(* Logix 5000 project; controller lab_1 vendor 1 type 14 code 96 rev 28.11; software revision 28.00 *)

TASK MainTask (continuous, watchdog 500 ms) : MainProgram

MODULES
   Local : vendor 1 type 14 code 96 (ICP 1, rev 28.11)
      INPUT : vendor 1 type 7 code 2 (ICP 2, rev 3.1, Input RPI 20 ms)
      RELAY_4 : 1756-OW16I (ICP 4, rev 3.1, Output RPI 20 ms)
      Relay_1 : 1756-OW16I (ICP 0, rev 3.3, Output RPI 20 ms)
      Relay_8 : 1756-IF6I (ICP 6, rev 1.1, Input RPI 100 ms)
      Relay_7 : vendor 1 type 10 code 4 (ICP 5, rev 1.12, Output RPI 25 ms)
END_MODULES

PROGRAM MainProgram   (* main routine MainRoutine *)
VAR
   BAND_01 : FBD_BOOLEAN_AND := (In1 := 1, In2 := 1, In3 := 1, In4 := 1, In5 := 1, In6 := 1, In7 := 1, In8 := 1);
   BOR_01 : FBD_BOOLEAN_OR;
   ESTOP : ALIAS FOR Local:2:I.Data.8;
   RED_LIGHT : ALIAS FOR Local:4:O.Data.2;
   run : BOOL;
   RUN_CMD : BOOL;
   START : ALIAS FOR Local:2:I.Data.0;
   STOP : ALIAS FOR Local:2:I.Data.9;
END_VAR

ROUTINE FBD_Motor_Control   (* function block diagram *)
   SHEET 1
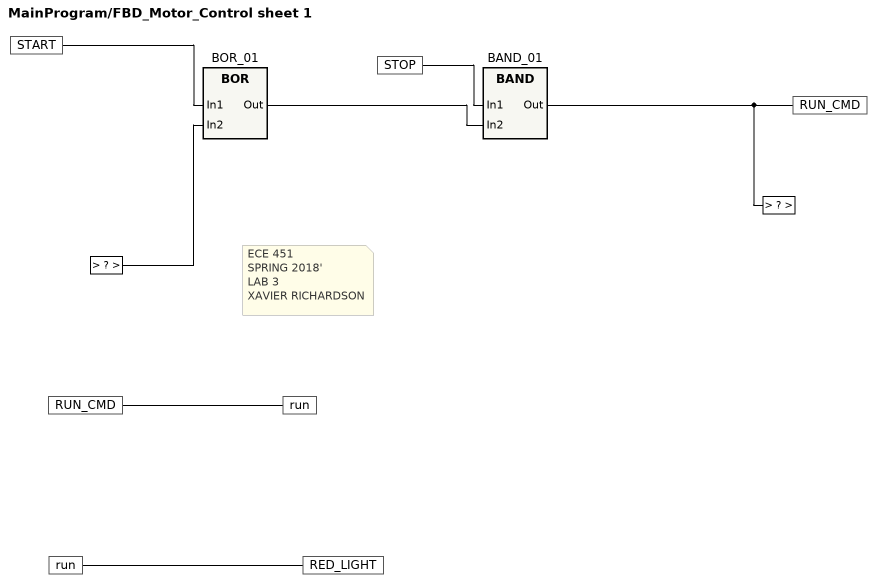
   // ECE 451
   // SPRING 2018'
   // LAB 3
   // XAVIER RICHARDSON
   BOR_01 : BOR(In1 := START, In2 := WIRE(?) {feedback});
   run := RUN_CMD;
   RED_LIGHT := run;
   BAND_01 : BAND(In1 := STOP, In2 := BOR_01.Out);
   WIRE(?) := BAND_01.Out;
   RUN_CMD := BAND_01.Out;
END_ROUTINE

ROUTINE MainRoutine   (* ladder *)
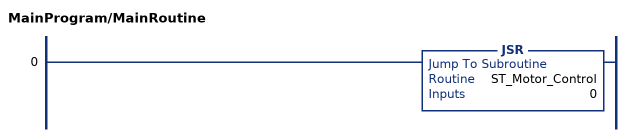
   0: JSR(ST_Motor_Control,0);
END_ROUTINE

ROUTINE Motor_Control   (* ladder *)
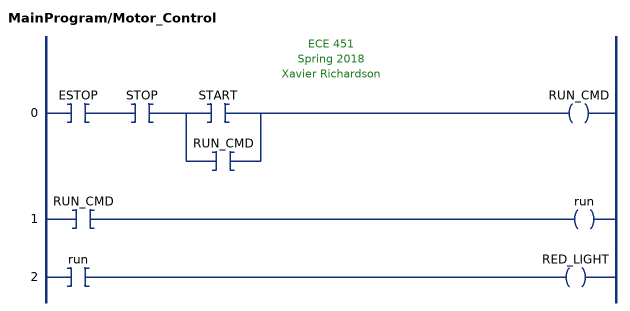
   // ECE 451
   // Spring 2018
   // Xavier Richardson
   0: XIC(ESTOP)XIC(STOP)[XIC(START) ,XIC(RUN_CMD) ]OTE(RUN_CMD);
   1: XIC(RUN_CMD)OTE(run);
   2: XIC(run)OTE(RED_LIGHT);
END_ROUTINE

ROUTINE ST_Motor_Control   (* structured text *)
   (*
   ECE 451 SPRING 2018
   XAVIER RICHARDSON
   *)
   
   //1ST RUNG
   
   RUN_CMD := (START or RUN_CMD) and STOP AND ESTOP;
   
   /////2ND RUNG
   
   run := RUN_CMD;
   
   ////////////3RD RUNG
   
   run := RED_LIGHT;
END_ROUTINE
END_PROGRAM
